# B&R Automation Studio project RobotLineDemo (part 2)

### BRRole.brrole - 5APC4100_TGL4_000/AccessAndSecurity/UserRoleSystem/BRRole.brrole
```
Element BR_Anonymous (Type=BRRole)
Element BR_Engineer (Type=BRRole)
Element BR_Observer (Type=BRRole)
Element BR_SafetyAdmin (Type=BRRole)
Element BR_SecurityAdmin (Type=BRRole)
```

- Physical/Config1/5APC4100_TGL4_000/IoMap.iom: same as Physical/Config1/5APC4100_TGL4_000/Cpu.per
- Physical/Config1/5APC4100_TGL4_000/PvMap.vvm: same as Physical/Config1/5APC4100_TGL4_000/Cpu.per
### Config.mappmotioncfg - 5APC4100_TGL4_000/mappMotion/Config.mappmotioncfg
```
Element MappMotionConfiguration (Type=mappmotioncfg)
  Logger:
    SelectiveLogging = Used
      AdministrativeCommands = Suppressed
      InformationalCommands = Suppressed
  Diagnostics:
    Snapshot = NotUsed
```

### ConvAxes.axis - 5APC4100_TGL4_000/mappMotion/Conveyors/ConvAxes.axis
```
Element gAxis_Conveyor_1 (Type=axis)
  BaseType = LinearPeriodic
    PeriodSettings:
      Period = 4000.0
  MovementLimits:
    Acceleration:
      Acceleration = 1000
    Deceleration:
      Deceleration = 1000
Element gAxis_Conveyor_2 (Type=axis)
  BaseType = LinearPeriodic
    PeriodSettings:
      Period = 4000.0
  MovementLimits:
    Acceleration:
      Acceleration = 1000
    Deceleration:
      Deceleration = 1000
```

### TrkPaths.trackingpath - 5APC4100_TGL4_000/mappMotion/Conveyors/TrkPaths.trackingpath
```
Element gTrkPath_Conveyor_1 (Type=trackingpath)
  Type:
    MaxTrackingFrames = 200
    MaxPositionError = 7.0
    MotionSource = Axis
      AxisRef = gAxis_Conveyor_1
    TrackingFrames:
      AutomaticCreation:
        Condition[1]:
          Distance = 150.0
          Activation = ProcessVariable
            ProcessVariableName = ::MovePrg:Cmd.Details.AutoCreationPath1
          Position:
            Translation:
              X = 0
              Y = -150
        Condition[2]:
          Distance = 150.0
          Activation = ProcessVariable
            ProcessVariableName = ::MovePrg:Cmd.Details.AutoCreationPath1
          Position:
            Translation:
              X = 0
              Y = -75
        Condition[3]:
          Distance = 150.0
          Activation = ProcessVariable
            ProcessVariableName = ::MovePrg:Cmd.Details.AutoCreationPath1
          Position:
            Translation:
              X = 0
              Y = 0
      AutomaticDeletion:
        Condition[1]:
          MinPosition = 0
          MaxPosition = 7000
        Condition[2] = AfterDesynchronization
          AxesGroupRef = gAxesGroup_D4r1100R_1
        Condition[3] = AfterDesynchronization
          AxesGroupRef = gAxesGroup_D4r1100R_2
        Condition[4] = AfterDesynchronization
          AxesGroupRef = gAxesGroup_D4r1100R_3
        Condition[5] = AfterDesynchronization
          AxesGroupRef = gAxesGroup_D4r1100R_4
        Condition[6] = AfterDesynchronization
          AxesGroupRef = gAxesGroup_D4r1100R_5
        Condition[7] = AfterDesynchronization
          AxesGroupRef = gAxesGroup_D4r1100R_6
  SceneViewerObject:
    Frame = Invisible
    Content:
      Template[1]:
        Name = Frame
      Template[2]:
        Name = Product
        VisualRepresentation = 3DMesh
          FileName = Product.tnr
          Material = LightGreyMatte
        Filter[1] = AttributeBased
          Type = ForbiddenBits
            Mask = 2#0000_0000_0000_0000_0000_0000_0000_0001
      Template[3]:
        Name = ProductSelected
        VisualRepresentation = 3DMesh
          FileName = Product.tnr
        Filter[1] = AttributeBased
          Type = MandatoryBits
            Mask = 2#0000_0000_0000_0000_0000_0000_0000_0001
Element gTrkPath_Conveyor_2 (Type=trackingpath)
  Type:
    MaxTrackingFrames = 200
    MaxPositionError = 7.0
    MotionSource = Axis
      AxisRef = gAxis_Conveyor_2
    TrackingFrames:
      AutomaticDeletion:
        Condition[1]:
          MinPosition = -200
          MaxPosition = 7800
  SceneViewerObject:
    Frame = Invisible
    Content:
      Template[1]:
        Name = Frame
      Template[2]:
        Name = Tray
        VisualRepresentation = 3DMesh
          FileName = Tray.tnr
          Material = LightGreyMatte
        Filter[1] = AttributeBased
          Type = MandatoryBits
            Mask = 2#0100_0000_0000
      Template[3]:
        Name = Product
        VisualRepresentation = 3DMesh
          FileName = Product.tnr
          Material = LightGreyMatte
        Filter[1] = AttributeBased
          Type = MandatoryBits
            Mask = 2#0000_0000_0000_0000_0000_1000_0000_0000
```

### Config_1.axesgroup - 5APC4100_TGL4_000/mappMotion/Robots/Codian_D4r1100R_1/Config_1.axesgroup
```
Element gAxesGroup_D4r1100R_1 (Type=axesgroup)  // Codian D4-ST41-1100-R30 [RobotID="CodianD4ST41r1100R30" Version="6.4.1"]
  Type = PathGenAxesGroup
    ProcessingTaskClass = 1
    PhysicalAxes:
      JointAxes:
        JointAxis[1]:
          AxisRef = gAxisQ1_D4r1100R_1
        JointAxis[2]:
          AxisRef = gAxisQ2_D4r1100R_1
        JointAxis[3]:
          AxisRef = gAxisQ3_D4r1100R_1
        JointAxis[4]:
          Name = QC
          AxisRef = gAxisQC_D4r1100R_1
    MechanicalSystem:
      MechSysRef = MechSys_D4r1100R_1
    BasicSettings:
      GeometryPlanning:
        Rounding:
          SymmetricRounding = No
          LastSegment = Whole
          AvoidZeroCurvature = Yes
          NonCartesianRounding = Yes
        MaxTangentialTransitionDeviation = 0.05
      TrajectoryPlanning:
        TorqueLimitConsideration = Approximation
      Miscellaneous:
        TimeStretchOverride:
          JerkSuppression = Basic
            AdaptationTime = 0.3
    StopReaction:
      AxisError:
        AxisReaction = DynamicStop
    AxesGroupFeatures:
      FeatureRef[1] = Feature_Programs_D4r1100R_1
      FeatureRef[2] = Feature_Jogging_D4r1100R_1
      FeatureRef[3] = Feature_FeedForward_D4r1100R_1
      FeatureRef[4] = FrameHierarchyRotBaseAngle1
      FeatureRef[5] = ToolSetup
      FeatureRef[6] = Tracking
      FeatureRef[7] = PathDefinitions
      FeatureRef[8] = Feature_TrkFrmSel_R1
```

### Config_2.axis - 5APC4100_TGL4_000/mappMotion/Robots/Codian_D4r1100R_1/Config_2.axis
```
Element gAxisQ1_D4r1100R_1 (Type=axis)  // Codian D4-ST41-1100-R30 [RobotID="CodianD4ST41r1100R30" Version="6.4.1"]
  BaseTypeIsReadOnly = 1
  BaseType = RotaryBounded
    MeasurementUnitIsReadOnly = 1
    MeasurementResolutionIsReadOnly = 1
    MeasurementResolution = 0.001
    CountDirectionIsReadOnly = 1
    CountDirection = Inverse
  MovementLimitsIsReadOnly = 1
  MovementLimits = InternalForPathControlledAxis
    Position:
      LowerLimitMin = -45.0
      UpperLimitMax = 103.0
      LowerLimit = -45.0
      UpperLimit = 103.0
    VelocityIsReadOnly = 1
    Velocity:
      VelocityMax = 410.0
      Velocity = 410.0
    AccelerationIsReadOnly = 1
    Acceleration:
      AccelerationMax = 25000.0
      Acceleration = 25000.0
    DecelerationIsReadOnly = 1
    Deceleration:
      DecelerationMax = 25000.0
      Deceleration = 25000.0
    JerkIsReadOnly = 1
    Jerk = Advanced
      JerkAccelerationPositiveMin = 0.0
      JerkAccelerationPositiveMax = 5000000.0
      JerkAccelerationPositive = 5000000.0
      JerkAccelerationNegativeMin = 0.0
      JerkAccelerationNegativeMax = 5000000.0
      JerkAccelerationNegative = 5000000.0
      JerkDecelerationPositiveMin = 0.0
      JerkDecelerationPositiveMax = 5000000.0
      JerkDecelerationPositive = 5000000.0
      JerkDecelerationNegativeMin = 0.0
      JerkDecelerationNegativeMax = 5000000.0
      JerkDecelerationNegative = 5000000.0
    TorqueIsReadOnly = 1
    Torque = Basic
      TorqueMax = 15.0
      Torque = 15.0
Element gAxisQ2_D4r1100R_1 (Type=axis)  // Codian D4-ST41-1100-R30 [RobotID="CodianD4ST41r1100R30" Version="6.4.1"]
  BaseTypeIsReadOnly = 1
  BaseType = RotaryBounded
    MeasurementUnitIsReadOnly = 1
    MeasurementResolutionIsReadOnly = 1
    MeasurementResolution = 0.001
    CountDirectionIsReadOnly = 1
    CountDirection = Inverse
  MovementLimitsIsReadOnly = 1
  MovementLimits = InternalForPathControlledAxis
    Position:
      LowerLimitMin = -45.0
      UpperLimitMax = 103.0
      LowerLimit = -45.0
      UpperLimit = 103.0
    VelocityIsReadOnly = 1
    Velocity:
      VelocityMax = 410.0
      Velocity = 410.0
    AccelerationIsReadOnly = 1
    Acceleration:
      AccelerationMax = 25000.0
      Acceleration = 25000.0
    DecelerationIsReadOnly = 1
    Deceleration:
      DecelerationMax = 25000.0
      Deceleration = 25000.0
    JerkIsReadOnly = 1
    Jerk = Advanced
      JerkAccelerationPositiveMin = 0.0
      JerkAccelerationPositiveMax = 5000000.0
      JerkAccelerationPositive = 5000000.0
      JerkAccelerationNegativeMin = 0.0
      JerkAccelerationNegativeMax = 5000000.0
      JerkAccelerationNegative = 5000000.0
      JerkDecelerationPositiveMin = 0.0
      JerkDecelerationPositiveMax = 5000000.0
      JerkDecelerationPositive = 5000000.0
      JerkDecelerationNegativeMin = 0.0
      JerkDecelerationNegativeMax = 5000000.0
      JerkDecelerationNegative = 5000000.0
    TorqueIsReadOnly = 1
    Torque = Basic
      TorqueMax = 15.0
      Torque = 15.0
Element gAxisQ3_D4r1100R_1 (Type=axis)  // Codian D4-ST41-1100-R30 [RobotID="CodianD4ST41r1100R30" Version="6.4.1"]
  BaseTypeIsReadOnly = 1
  BaseType = RotaryBounded
    MeasurementUnitIsReadOnly = 1
    MeasurementResolutionIsReadOnly = 1
    MeasurementResolution = 0.001
    CountDirectionIsReadOnly = 1
    CountDirection = Inverse
  MovementLimitsIsReadOnly = 1
  MovementLimits = InternalForPathControlledAxis
    Position:
      LowerLimitMin = -45.0
      UpperLimitMax = 103.0
      LowerLimit = -45.0
      UpperLimit = 103.0
    VelocityIsReadOnly = 1
    Velocity:
      VelocityMax = 410.0
      Velocity = 410.0
    AccelerationIsReadOnly = 1
    Acceleration:
      AccelerationMax = 25000.0
      Acceleration = 25000.0
    DecelerationIsReadOnly = 1
    Deceleration:
      DecelerationMax = 25000.0
      Deceleration = 25000.0
    JerkIsReadOnly = 1
    Jerk = Advanced
      JerkAccelerationPositiveMin = 0.0
      JerkAccelerationPositiveMax = 5000000.0
      JerkAccelerationPositive = 5000000.0
      JerkAccelerationNegativeMin = 0.0
      JerkAccelerationNegativeMax = 5000000.0
      JerkAccelerationNegative = 5000000.0
      JerkDecelerationPositiveMin = 0.0
      JerkDecelerationPositiveMax = 5000000.0
      JerkDecelerationPositive = 5000000.0
      JerkDecelerationNegativeMin = 0.0
      JerkDecelerationNegativeMax = 5000000.0
      JerkDecelerationNegative = 5000000.0
    TorqueIsReadOnly = 1
    Torque = Basic
      TorqueMax = 15.0
      Torque = 15.0
Element gAxisQC_D4r1100R_1 (Type=axis)  // Codian D4-ST41-1100-R30 [RobotID="CodianD4ST41r1100R30" Version="6.4.1"]
  BaseTypeIsReadOnly = 1
  BaseType = Rotary
    MeasurementUnitIsReadOnly = 1
    MeasurementResolutionIsReadOnly = 1
    MeasurementResolution = 0.001
    CountDirectionIsReadOnly = 1
  MovementLimitsIsReadOnly = 1
  MovementLimits = InternalForPathControlledAxis
    VelocityIsReadOnly = 1
    Velocity:
      VelocityMax = 1150.0
      Velocity = 1150.0
    AccelerationIsReadOnly = 1
    Acceleration:
      AccelerationMax = 28000.0
      Acceleration = 28000.0
    DecelerationIsReadOnly = 1
    Deceleration:
      DecelerationMax = 28000.0
      Deceleration = 28000.0
    JerkIsReadOnly = 1
    Jerk = Advanced
      JerkAccelerationPositiveMin = 0.0
      JerkAccelerationPositiveMax = 4000000.0
      JerkAccelerationPositive = 4000000.0
      JerkAccelerationNegativeMin = 0.0
      JerkAccelerationNegativeMax = 4000000.0
      JerkAccelerationNegative = 4000000.0
      JerkDecelerationPositiveMin = 0.0
      JerkDecelerationPositiveMax = 4000000.0
      JerkDecelerationPositive = 4000000.0
      JerkDecelerationNegativeMin = 0.0
      JerkDecelerationNegativeMax = 4000000.0
      JerkDecelerationNegative = 4000000.0
    TorqueIsReadOnly = 1
    Torque = Basic
      TorqueMax = 9.0
      Torque = 9.0
```

### Config_3.mechanicalsystem - 5APC4100_TGL4_000/mappMotion/Robots/Codian_D4r1100R_1/Config_3.mechanicalsystem
```
Element MechSys_D4r1100R_1 (Type=mechanicalsystem)  // Codian D4-ST41-1100-R30 [RobotID="CodianD4ST41r1100R30" Version="6.4.1"]
  TypeIsReadOnly = 1
  Type = Delta
    SubtypeIsReadOnly = 1
    Subtype = 4AxesDeltaA
      SceneViewerObject = ObjectID
        ID = 2540
      DescriptionIsReadOnly = 1
      Description:
        Dimensions:
          BasePlatform:
            ArmLinkPointIsReadOnly = 1
            Arm1LinkPoint:
              Radius = 207.5
              Z = -110.0
            Arm2LinkPoint:
              Angle = -120.0
              Radius = 207.5
              Z = -110.0
            Arm3LinkPoint:
              Angle = -240.0
              Radius = 207.5
              Z = -110.0
          Arms:
            ArmIsReadOnly = 1
            Arm1:
              UpperArmLength = 320.0
              LowerArmLength = 850.0
            Arm2:
              UpperArmLength = 320.0
              LowerArmLength = 850.0
            Arm3:
              UpperArmLength = 320.0
              LowerArmLength = 850.0
            LowerArmPairDistance = 154.0
          EndEffectorPlatform:
            ArmLinkPointIsReadOnly = 1
            Arm1LinkPoint:
              Radius = 70.0
            Arm2LinkPoint:
              Radius = 70.0
            Arm3LinkPoint:
              Radius = 70.0
            TranslationToFlange:
              Z = -59.0
        Offsets:
          JointAxisIsReadOnly = 1
          JointAxis[1]
          JointAxis[2]
          JointAxis[3]
          JointAxis[4]
        CountDirections:
          JointAxisIsReadOnly = 1
          JointAxis[1]
          JointAxis[2]
          JointAxis[3]
          JointAxis[4]
      TcpOrientation:
        Frames = Used
      WireFrameModel:
        UpperArm1:
          Distance = 5
        LowerArm1:
          Distance = 5
        UpperArm2:
          Distance = 5
        LowerArm2:
          Distance = 5
        UpperArm3:
          Distance = 5
        LowerArm3:
          Distance = 5
        EndEffectorPlatformToFlange:
          Distance = 5
        FlangeToTcp = NotUsed
      DynamicModelIsReadOnly = 1
      InternalDynamicModelIsReadOnly = 1
      InternalDynamicModel = Used
        TypeIsReadOnly = 1
        Type = Codian D4-ST41-1100-R30
        Row[1]:
          Value = 4
          Unit = Variant
          Description = Type of dynamic model
        Row[2]:
          Index = 1
          Value = 2.739
          Unit = 
          Description = m1
        Row[3]:
          Index = 2
          Value = 0.2990988
          Unit = 
          Description = m1*rc1x
        Row[4]:
          Index = 3
          Unit = 
          Description = m1*rc1y
        Row[5]:
          Index = 4
          Value = 0.0257466
          Unit = 
          Description = m1*rc1z
        Row[6]:
          Index = 5
          Unit = 
          Description = m1*rc1x*rc1y
        Row[7]:
          Index = 6
          Unit = 
          Description = m1*rc1y*rc1z
        Row[8]:
          Index = 7
          Value = 0.00281152872
          Unit = 
          Description = m1*rc1x*rc1z
        Row[9]:
          Index = 8
          Value = 0.03266158896
          Unit = 
          Description = m1*rc1x^2
        Row[10]:
          Index = 9
          Unit = 
          Description = m1*rc1y^2
        Row[11]:
          Index = 10
          Value = 0.00024201804
          Unit = 
          Description = m1*rc1z^2
        Row[12]:
          Index = 11
          Unit = 
          Description = Jxx1
        Row[13]:
          Index = 12
          Value = 0.0423
          Unit = 
          Description = Jyy1
        Row[14]:
          Index = 13
          Unit = 
          Description = Jzz1
        Row[15]:
          Index = 14
          Value = 2.739
          Unit = 
          Description = m2
        Row[16]:
          Index = 15
          Value = 0.2990988
          Unit = 
          Description = m2*rc2x
        Row[17]:
          Index = 16
          Unit = 
          Description = m2*rc2y
        Row[18]:
          Index = 17
          Value = 0.0257466
          Unit = 
          Description = m2*rc2z
        Row[19]:
          Index = 18
          Unit = 
          Description = m2*rc2x*rc2y
        Row[20]:
          Index = 19
          Unit = 
          Description = m2*rc2y*rc2z
        Row[21]:
          Index = 20
          Value = 0.00281152872
          Unit = 
          Description = m2*rc2x*rc2z
        Row[22]:
          Index = 21
          Value = 0.03266158896
          Unit = 
          Description = m2*rc2x^2
        Row[23]:
          Index = 22
          Unit = 
          Description = m2*rc2y^2
        Row[24]:
          Index = 23
          Value = 0.00024201804
          Unit = 
          Description = m2*rc2z^2
        Row[25]:
          Index = 24
          Unit = 
          Description = Jxx2
        Row[26]:
          Index = 25
          Value = 0.0423
          Unit = 
          Description = Jyy2
        Row[27]:
          Index = 26
          Unit = 
          Description = Jzz2
        Row[28]:
          Index = 27
          Value = 2.739
          Unit = 
          Description = m3
        Row[29]:
          Index = 28
          Value = 0.2990988
          Unit = 
          Description = m3*rc3x
        Row[30]:
          Index = 29
          Unit = 
          Description = m3*rc3y
        Row[31]:
          Index = 30
          Value = 0.0257466
          Unit = 
          Description = m3*rc3z
        Row[32]:
          Index = 31
          Unit = 
          Description = m3*rc3x*rc3y
        Row[33]:
          Index = 32
          Unit = 
          Description = m3*rc3y*rc3z
        Row[34]:
          Index = 33
          Value = 0.00281152872
          Unit = 
          Description = m3*rc3x*rc3z
        Row[35]:
          Index = 34
          Value = 0.03266158896
          Unit = 
          Description = m3*rc3x^2
        Row[36]:
          Index = 35
          Unit = 
          Description = m3*rc3y^2
        Row[37]:
          Index = 36
          Value = 0.00024201804
          Unit = 
          Description = m3*rc3z^2
        Row[38]:
          Index = 37
          Unit = 
          Description = Jxx3
        Row[39]:
          Index = 38
          Value = 0.0423
          Unit = 
          Description = Jyy3
        Row[40]:
          Index = 39
          Unit = 
          Description = Jzz3
        Row[41]:
          Index = 40
          Value = 0.808
          Unit = 
          Description = m4
        Row[42]:
          Index = 41
          Unit = 
          Description = m4*rc4x
        Row[43]:
          Index = 42
          Unit = 
          Description = m4*rc4y
        Row[44]:
          Index = 43
          Unit = 
          Description = m4*rc4z
        Row[45]:
          Index = 44
          Unit = 
          Description = m4*rc4x*rc4y
        Row[46]:
          Index = 45
          Unit = 
          Description = m4*rc4y*rc4z
        Row[47]:
          Index = 46
          Unit = 
          Description = m4*rc4x*rc4z
        Row[48]:
          Index = 47
          Unit = 
          Description = m4*rc4x^2
        Row[49]:
          Index = 48
          Unit = 
          Description = m4*rc4y^2
        Row[50]:
          Index = 49
          Unit = 
          Description = m4*rc4z^2
        Row[51]:
          Index = 50
          Value = 0.0901
          Unit = 
          Description = Jxx4
        Row[52]:
          Index = 51
          Value = 0.0901
          Unit = 
          Description = Jyy4
        Row[53]:
          Index = 52
          Unit = 
          Description = Jzz4
        Row[54]:
          Index = 53
          Value = 0.808
          Unit = 
          Description = m5
        Row[55]:
          Index = 54
          Unit = 
          Description = m5*rc5x
        Row[56]:
          Index = 55
          Unit = 
          Description = m5*rc5y
        Row[57]:
          Index = 56
          Unit = 
          Description = m5*rc5z
        Row[58]:
          Index = 57
          Unit = 
          Description = m5*rc5x*rc5y
        Row[59]:
          Index = 58
          Unit = 
          Description = m5*rc5y*rc5z
        Row[60]:
          Index = 59
          Unit = 
          Description = m5*rc5x*rc5z
        Row[61]:
          Index = 60
          Unit = 
          Description = m5*rc5x^2
        Row[62]:
          Index = 61
          Unit = 
          Description = m5*rc5y^2
        Row[63]:
          Index = 62
          Unit = 
          Description = m5*rc5z^2
        Row[64]:
          Index = 63
          Value = 0.0901
          Unit = 
          Description = Jxx5
        Row[65]:
          Index = 64
          Value = 0.0901
          Unit = 
          Description = Jyy5
        Row[66]:
          Index = 65
          Unit = 
          Description = Jzz5
        Row[67]:
          Index = 66
          Value = 0.808
          Unit = 
          Description = m6
        Row[68]:
          Index = 67
          Unit = 
          Description = m6*rc6x
        Row[69]:
          Index = 68
          Unit = 
          Description = m6*rc6y
        Row[70]:
          Index = 69
          Unit = 
          Description = m6*rc6z
        Row[71]:
          Index = 70
          Unit = 
          Description = m6*rc6x*rc6y
        Row[72]:
          Index = 71
          Unit = 
          Description = m6*rc6y*rc6z
        Row[73]:
          Index = 72
          Unit = 
          Description = m6*rc6x*rc6z
        Row[74]:
          Index = 73
          Unit = 
          Description = m6*rc6x^2
        Row[75]:
          Index = 74
          Unit = 
          Description = m6*rc6y^2
        Row[76]:
          Index = 75
          Unit = 
          Description = m6*rc6z^2
        Row[77]:
          Index = 76
          Value = 0.0901
          Unit = 
          Description = Jxx6
        Row[78]:
          Index = 77
          Value = 0.0901
          Unit = 
          Description = Jyy6
        Row[79]:
          Index = 78
          Unit = 
          Description = Jzz6
        Row[80]:
          Index = 79
          Value = 2.005
          Unit = 
          Description = m7
        Row[81]:
          Index = 80
          Unit = 
          Description = m7*rc7x
        Row[82]:
          Index = 81
          Unit = 
          Description = m7*rc7y
        Row[83]:
          Index = 82
          Value = 0.47159605
          Unit = 
          Description = m7*rc7z
        Row[84]:
          Index = 83
          Unit = 
          Description = m7*rc7x*rc7y
        Row[85]:
          Index = 84
          Unit = 
          Description = m7*rc7y*rc7z
        Row[86]:
          Index = 85
          Unit = 
          Description = m7*rc7x*rc7z
        Row[87]:
          Index = 86
          Unit = 
          Description = m7*rc7x^2
        Row[88]:
          Index = 87
          Unit = 
          Description = m7*rc7y^2
        Row[89]:
          Index = 88
          Value = 0.110924106921
          Unit = 
          Description = m7*rc7z^2
        Row[90]:
          Index = 89
          Value = 0.071421443
          Unit = 
          Description = Jxx7
        Row[91]:
          Index = 90
          Value = 0.071421443
          Unit = 
          Description = Jyy7
        Row[92]:
          Index = 91
          Value = 0.0003844
          Unit = 
          Description = Jzz7
        Row[93]:
          Index = 92
          Value = 1.8
          Unit = 
          Description = m8
        Row[94]:
          Index = 93
          Unit = 
          Description = m8*rc8x
        Row[95]:
          Index = 94
          Unit = 
          Description = m8*rc8y
        Row[96]:
          Index = 95
          Value = 0.520488
          Unit = 
          Description = m8*rc8z
        Row[97]:
          Index = 96
          Unit = 
          Description = m8*rc8x*rc8y
        Row[98]:
          Index = 97
          Unit = 
          Description = m8*rc8y*rc8z
        Row[99]:
          Index = 98
          Unit = 
          Description = m8*rc8x*rc8z
        Row[100]:
          Index = 99
          Unit = 
          Description = m8*rc8x^2
        Row[101]:
          Index = 100
          Unit = 
          Description = m8*rc8y^2
        Row[102]:
          Index = 101
          Value = 0.15050431008
          Unit = 
          Description = m8*rc8z^2
        Row[103]:
          Index = 102
          Value = 0.093006951
          Unit = 
          Description = Jxx8
        Row[104]:
          Index = 103
          Value = 0.093006951
          Unit = 
          Description = Jyy8
        Row[105]:
          Index = 104
          Value = 0.00097
          Unit = 
          Description = Jzz8
        Row[106]:
          Index = 105
          Value = 2.094
          Unit = 
          Description = m9
        Row[107]:
          Index = 106
          Unit = 
          Description = m9*rc9x
        Row[108]:
          Index = 107
          Unit = 
          Description = m9*rc9y
        Row[109]:
          Index = 108
          Unit = 
          Description = m9*rc9z
        Row[110]:
          Index = 109
          Unit = 
          Description = m9*rc9x*rc9y
        Row[111]:
          Index = 110
          Unit = 
          Description = m9*rc9y*rc9z
        Row[112]:
          Index = 111
          Unit = 
          Description = m9*rc9x*rc9z
        Row[113]:
          Index = 112
          Unit = 
          Description = m9*rc9x^2
        Row[114]:
          Index = 113
          Unit = 
          Description = m9*rc9y^2
        Row[115]:
          Index = 114
          Unit = 
          Description = m9*rc9z^2
        Row[116]:
          Index = 115
          Unit = 
          Description = Jxx9
        Row[117]:
          Index = 116
          Unit = 
          Description = Jyy9
        Row[118]:
          Index = 117
          Unit = 
          Description = Jzz9
        Row[119]:
          Index = 118
          Unit = 
          Description = m10
        Row[120]:
          Index = 119
          Unit = 
          Description = m10*rc10x
        Row[121]:
          Index = 120
          Unit = 
          Description = m10*rc10y
        Row[122]:
          Index = 121
          Unit = 
          Description = m10*rc10z
        Row[123]:
          Index = 122
          Unit = 
          Description = m10*rc10x*rc10y
        Row[124]:
          Index = 123
          Unit = 
          Description = m10*rc10y*rc10z
        Row[125]:
          Index = 124
          Unit = 
          Description = m10*rc10x*rc10z
        Row[126]:
          Index = 125
          Unit = 
          Description = m10*rc10x^2
        Row[127]:
          Index = 126
          Unit = 
          Description = m10*rc10y^2
        Row[128]:
          Index = 127
          Unit = 
          Description = m10*rc10z^2
        Row[129]:
          Index = 128
          Unit = 
          Description = Jxx10
        Row[130]:
          Index = 129
          Unit = 
          Description = Jyy10
        Row[131]:
          Index = 130
          Value = 0.0001507
          Unit = 
          Description = Jzz10
        Row[132]:
          Index = 144
          Value = 0.0005703
          Unit = 
          Description = JDrive1
        Row[133]:
          Index = 145
          Value = 0.0005703
          Unit = 
          Description = JDrive2
        Row[134]:
          Index = 146
          Value = 0.0005703
          Unit = 
          Description = JDrive3
        Row[135]:
          Index = 147
          Value = 0.0001462
          Unit = 
          Description = JDrive4
        Row[136]:
          Index = 148
          Value = 2.35907414398
          Unit = 
          Description = dV1
        Row[137]:
          Index = 149
          Value = 2.35907414398
          Unit = 
          Description = dV2
        Row[138]:
          Index = 150
          Value = 2.35907414398
          Unit = 
          Description = dV3
        Row[139]:
          Index = 151
          Value = 0.0159154943092
          Unit = 
          Description = dV4
        Row[140]:
          Index = 152
          Value = 4.235
          Unit = 
          Description = dC1
        Row[141]:
          Index = 153
          Value = 4.235
          Unit = 
          Description = dC2
        Row[142]:
          Index = 154
          Value = 4.235
          Unit = 
          Description = dC3
        Row[143]:
          Index = 155
          Value = 1.0
          Unit = 
          Description = dC4
      InternalDynamicLimits = Used
        TypeIsReadOnly = 1
        Type = Codian D4-ST41-1100-R30
        GearboxLimits:
          Row[1]:
            Value = 4
            Unit = Variant
            Description = Type of dynamic model
          Row[2]:
            Index = 1
            Value = 370.0
            Unit = Nm
            Description = Gearbox Drive 1 Output Torque Limit
          Row[3]:
            Index = 2
            Value = 370.0
            Unit = Nm
            Description = Gearbox Drive 2 Output Torque Limit
          Row[4]:
            Index = 3
            Value = 370.0
            Unit = Nm
            Description = Gearbox Drive 3 Output Torque Limit
          Row[5]:
            Index = 4
            Value = 17.0
            Unit = Nm
            Description = Gearbox Drive 4 Output Torque Limit
        CrossSectionLimits:
          Row[1]:
            Value = 4
            Unit = Variant
            Description = Type of dynamic model
          Row[2]:
            Index = 1
            Value = 10000.0
            Unit = N
            Description = 
          Row[3]:
            Index = 2
            Value = 10000.0
            Unit = N
            Description = 
          Row[4]:
            Index = 3
            Value = 10000.0
            Unit = N
            Description = 
          Row[5]:
            Index = 4
            Value = 141.0
            Unit = Nm
            Description = 
          Row[6]:
            Index = 5
            Value = 141.0
            Unit = Nm
            Description = 
          Row[7]:
            Index = 6
            Value = 10000.0
            Unit = Nm
            Description = 
          Row[8]:
            Index = 7
            Value = 750.0
            Unit = N
            Description = 
          Row[9]:
            Index = 8
            Value = 750.0
            Unit = N
            Description = 
          Row[10]:
            Index = 9
            Value = 750.0
            Unit = N
            Description = 
          Row[11]:
            Index = 10
            Value = 750.0
            Unit = N
            Description = 
          Row[12]:
            Index = 11
            Value = 750.0
            Unit = N
            Description = 
          Row[13]:
            Index = 12
            Value = 750.0
            Unit = N
            Description = 
      LoadDependentJerkLimitsIsReadOnly = 1
      LoadDependentJerkLimits = PayloadDependentJerkReduction
        JerkReduction[1]:
          PayloadInKgIsReadOnly = 1
          PayloadInKg = 0.0
          JerkReductionInPercentIsReadOnly = 1
          JerkReductionInPercent = 0.0
        JerkReduction[2]:
          PayloadInKgIsReadOnly = 1
          PayloadInKg = 7.0
          JerkReductionInPercentIsReadOnly = 1
          JerkReductionInPercent = 20.0
        JerkReduction[3]:
          PayloadInKgIsReadOnly = 1
          PayloadInKg = 13.0
          JerkReductionInPercentIsReadOnly = 1
          JerkReductionInPercent = 60.0
        JerkReduction[4]:
          PayloadInKgIsReadOnly = 1
          PayloadInKg = 19.0
          JerkReductionInPercentIsReadOnly = 1
          JerkReductionInPercent = 60.0
        JerkReduction[5]:
          PayloadInKgIsReadOnly = 1
          PayloadInKg = 23.0
          JerkReductionInPercentIsReadOnly = 1
          JerkReductionInPercent = 80.0
      JointAxesPositionLimits:
        JointAxisIsReadOnly = 1
        JointAxis[1]
        JointAxis[2]
        JointAxis[3]
        JointAxis[4]
      WorkingRangeIsReadOnly = 1
      WorkingRange = Extended
        MainCylinderDiameterIsReadOnly = 1
        MainCylinderDiameter = 1100.0
        BaseToTopConeIsReadOnly = 1
        BaseToTopCone = 735.0
        MainCylinderOffsetIsReadOnly = 1
        MainCylinderOffset = 270.0
        MainConeOffsetIsReadOnly = 1
        MainConeOffset = 350.0
        BottomConeOffsetIsReadOnly = 1
        BottomConeOffset = 420.0
        MainConeDiameterIsReadOnly = 1
        MainConeDiameter = 820.0
        BottomConeDiameterIsReadOnly = 1
        BottomConeDiameter = 340.0
        TopConeOffsetIsReadOnly = 1
        TopConeDiameterIsReadOnly = 1
        TopConeDiameter = 1100.0
```

### Config_4.axesgroupfeature - 5APC4100_TGL4_000/mappMotion/Robots/Codian_D4r1100R_1/Config_4.axesgroupfeature
```
Element Feature_TrkFrmSel_R1 (Type=axesgroupfeature)
  Type = TrackingFrameSelection
    Selectors:
      Selector[1]:
        Name = ProductSelector
        Strategy = MinimumDistanceToPoint
          Origin = MCS
            Translation:
              X = -350
              Y = 300
        Filters:
          Filter[1]:
            TrackingPathRef[1] = gTrkPath_Conveyor_1
          Filter[2] = SelectionArea
            Area[1] = Cylinder
              Origin = MCS
              Translation:
                X = -470
                Z = -100
              Dimensions:
                Radius = 475
                Height = 250
        LockingAfterSelection = AllSelectors
      Selector[2]:
        Name = PlacePositionSelector
        Strategy = MaximumXValueOnTrackingPath
        Filters:
          Filter[1]:
            TrackingPathRef[1] = gTrkPath_Conveyor_2
          Filter[2] = SelectionArea
            Area[1] = Cylinder
              Origin = MCS
              Translation:
                X = 250
                Z = -100
              Dimensions:
                Radius = 500
                Height = 250
        LockingAfterSelection = AllSelectors
      Selector[3]:
        Name = PlacePositionSelectorPrior
        Strategy = MaximumXValueOnTrackingPath
        Filters:
          Filter[1]:
            TrackingPathRef[1] = gTrkPath_Conveyor_2
          Filter[2] = SelectionArea
            Area[1]:
              Origin = MCS
              Translation:
                X = -300
                Y = 200
                Z = -100
              Dimensions:
                Length = 700
                Width = 200
                Height = 250
        LockingAfterSelection = AllSelectors
Element Feature_Programs_D4r1100R_1 (Type=axesgroupfeature)  // Codian D4-ST41-1100-R30 [RobotID="CodianD4ST41r1100R30" Version="6.4.1"]
  Type:
    InitialSettings:
      AccuracyHoldDelays = User defined
        UserAxesDelay = 0.06
    ProgramElements:
      PVs:
        PV[1]:
          PvName = ::MovePrg:GripperRobot1OpenClose
          Advanced:
            Alias = CloseGripper
            Synchronization = Path
Element Feature_Jogging_D4r1100R_1 (Type=axesgroupfeature)  // Codian D4-ST41-1100-R30 [RobotID="CodianD4ST41r1100R30" Version="6.4.1"]
  Type = Jogging
Element Feature_FeedForward_D4r1100R_1 (Type=axesgroupfeature)  // Codian D4-ST41-1100-R30 [RobotID="CodianD4ST41r1100R30" Version="6.4.1"]
  Type = FeedForward
    RiseTime = 0.25
    Filter = AxisJerkTime
```

### Config_5.axesgroup - 5APC4100_TGL4_000/mappMotion/Robots/Codian_D4r1100R_2/Config_5.axesgroup
```
Element gAxesGroup_D4r1100R_2 (Type=axesgroup)  // Codian D4-ST41-1100-R30 [RobotID="CodianD4ST41r1100R30" Version="6.4.1"]
  Type = PathGenAxesGroup
    ProcessingTaskClass = 1
    PhysicalAxes:
      JointAxes:
        JointAxis[1]:
          AxisRef = gAxisQ1_D4r1100R_2
        JointAxis[2]:
          AxisRef = gAxisQ2_D4r1100R_2
        JointAxis[3]:
          AxisRef = gAxisQ3_D4r1100R_2
        JointAxis[4]:
          Name = QC
          AxisRef = gAxisQC_D4r1100R_2
    MechanicalSystem:
      MechSysRef = MechSys_D4r1100R_2
    BasicSettings:
      GeometryPlanning:
        Rounding:
          SymmetricRounding = No
          LastSegment = Whole
          AvoidZeroCurvature = Yes
          NonCartesianRounding = Yes
        MaxTangentialTransitionDeviation = 0.05
      TrajectoryPlanning:
        TorqueLimitConsideration = Approximation
      Miscellaneous:
        TimeStretchOverride:
          JerkSuppression = Basic
            AdaptationTime = 0.3
    StopReaction:
      AxisError:
        AxisReaction = DynamicStop
    AxesGroupFeatures:
      FeatureRef[1] = Feature_Programs_D4r1100R_2
      FeatureRef[2] = Feature_Jogging_D4r1100R_2
      FeatureRef[3] = Feature_FeedForward_D4r1100R_2
      FeatureRef[4] = FrameHierarchyRotBaseAngle2
      FeatureRef[5] = ToolSetup
      FeatureRef[6] = Tracking
      FeatureRef[7] = PathDefinitions
      FeatureRef[8] = Feature_TrkFrmSel_R2
```

### Config_6.axis - 5APC4100_TGL4_000/mappMotion/Robots/Codian_D4r1100R_2/Config_6.axis
```
Element gAxisQ1_D4r1100R_2 (Type=axis)  // Codian D4-ST41-1100-R30 [RobotID="CodianD4ST41r1100R30" Version="6.4.1"]
  BaseTypeIsReadOnly = 1
  BaseType = RotaryBounded
    MeasurementUnitIsReadOnly = 1
    MeasurementResolutionIsReadOnly = 1
    MeasurementResolution = 0.001
    CountDirectionIsReadOnly = 1
    CountDirection = Inverse
  MovementLimitsIsReadOnly = 1
  MovementLimits = InternalForPathControlledAxis
    Position:
      LowerLimitMin = -45.0
      UpperLimitMax = 103.0
      LowerLimit = -45.0
      UpperLimit = 103.0
    VelocityIsReadOnly = 1
    Velocity:
      VelocityMax = 410.0
      Velocity = 410.0
    AccelerationIsReadOnly = 1
    Acceleration:
      AccelerationMax = 25000.0
      Acceleration = 25000.0
    DecelerationIsReadOnly = 1
    Deceleration:
      DecelerationMax = 25000.0
      Deceleration = 25000.0
    JerkIsReadOnly = 1
    Jerk = Advanced
      JerkAccelerationPositiveMin = 0.0
      JerkAccelerationPositiveMax = 5000000.0
      JerkAccelerationPositive = 5000000.0
      JerkAccelerationNegativeMin = 0.0
      JerkAccelerationNegativeMax = 5000000.0
      JerkAccelerationNegative = 5000000.0
      JerkDecelerationPositiveMin = 0.0
      JerkDecelerationPositiveMax = 5000000.0
      JerkDecelerationPositive = 5000000.0
      JerkDecelerationNegativeMin = 0.0
      JerkDecelerationNegativeMax = 5000000.0
      JerkDecelerationNegative = 5000000.0
    TorqueIsReadOnly = 1
    Torque = Basic
      TorqueMax = 15.0
      Torque = 15.0
Element gAxisQ2_D4r1100R_2 (Type=axis)  // Codian D4-ST41-1100-R30 [RobotID="CodianD4ST41r1100R30" Version="6.4.1"]
  BaseTypeIsReadOnly = 1
  BaseType = RotaryBounded
    MeasurementUnitIsReadOnly = 1
    MeasurementResolutionIsReadOnly = 1
    MeasurementResolution = 0.001
    CountDirectionIsReadOnly = 1
    CountDirection = Inverse
  MovementLimitsIsReadOnly = 1
  MovementLimits = InternalForPathControlledAxis
    Position:
      LowerLimitMin = -45.0
      UpperLimitMax = 103.0
      LowerLimit = -45.0
      UpperLimit = 103.0
    VelocityIsReadOnly = 1
    Velocity:
      VelocityMax = 410.0
      Velocity = 410.0
    AccelerationIsReadOnly = 1
    Acceleration:
      AccelerationMax = 25000.0
      Acceleration = 25000.0
    DecelerationIsReadOnly = 1
    Deceleration:
      DecelerationMax = 25000.0
      Deceleration = 25000.0
    JerkIsReadOnly = 1
    Jerk = Advanced
      JerkAccelerationPositiveMin = 0.0
      JerkAccelerationPositiveMax = 5000000.0
      JerkAccelerationPositive = 5000000.0
      JerkAccelerationNegativeMin = 0.0
      JerkAccelerationNegativeMax = 5000000.0
      JerkAccelerationNegative = 5000000.0
      JerkDecelerationPositiveMin = 0.0
      JerkDecelerationPositiveMax = 5000000.0
      JerkDecelerationPositive = 5000000.0
      JerkDecelerationNegativeMin = 0.0
      JerkDecelerationNegativeMax = 5000000.0
      JerkDecelerationNegative = 5000000.0
    TorqueIsReadOnly = 1
    Torque = Basic
      TorqueMax = 15.0
      Torque = 15.0
Element gAxisQ3_D4r1100R_2 (Type=axis)  // Codian D4-ST41-1100-R30 [RobotID="CodianD4ST41r1100R30" Version="6.4.1"]
  BaseTypeIsReadOnly = 1
  BaseType = RotaryBounded
    MeasurementUnitIsReadOnly = 1
    MeasurementResolutionIsReadOnly = 1
    MeasurementResolution = 0.001
    CountDirectionIsReadOnly = 1
    CountDirection = Inverse
  MovementLimitsIsReadOnly = 1
  MovementLimits = InternalForPathControlledAxis
    Position:
      LowerLimitMin = -45.0
      UpperLimitMax = 103.0
      LowerLimit = -45.0
      UpperLimit = 103.0
    VelocityIsReadOnly = 1
    Velocity:
      VelocityMax = 410.0
      Velocity = 410.0
    AccelerationIsReadOnly = 1
    Acceleration:
      AccelerationMax = 25000.0
      Acceleration = 25000.0
    DecelerationIsReadOnly = 1
    Deceleration:
      DecelerationMax = 25000.0
      Deceleration = 25000.0
    JerkIsReadOnly = 1
    Jerk = Advanced
      JerkAccelerationPositiveMin = 0.0
      JerkAccelerationPositiveMax = 5000000.0
      JerkAccelerationPositive = 5000000.0
      JerkAccelerationNegativeMin = 0.0
      JerkAccelerationNegativeMax = 5000000.0
      JerkAccelerationNegative = 5000000.0
      JerkDecelerationPositiveMin = 0.0
      JerkDecelerationPositiveMax = 5000000.0
      JerkDecelerationPositive = 5000000.0
      JerkDecelerationNegativeMin = 0.0
      JerkDecelerationNegativeMax = 5000000.0
      JerkDecelerationNegative = 5000000.0
    TorqueIsReadOnly = 1
    Torque = Basic
      TorqueMax = 15.0
      Torque = 15.0
Element gAxisQC_D4r1100R_2 (Type=axis)  // Codian D4-ST41-1100-R30 [RobotID="CodianD4ST41r1100R30" Version="6.4.1"]
  BaseTypeIsReadOnly = 1
  BaseType = Rotary
    MeasurementUnitIsReadOnly = 1
    MeasurementResolutionIsReadOnly = 1
    MeasurementResolution = 0.001
    CountDirectionIsReadOnly = 1
  MovementLimitsIsReadOnly = 1
  MovementLimits = InternalForPathControlledAxis
    VelocityIsReadOnly = 1
    Velocity:
      VelocityMax = 1150.0
      Velocity = 1150.0
    AccelerationIsReadOnly = 1
    Acceleration:
      AccelerationMax = 28000.0
      Acceleration = 28000.0
    DecelerationIsReadOnly = 1
    Deceleration:
      DecelerationMax = 28000.0
      Deceleration = 28000.0
    JerkIsReadOnly = 1
    Jerk = Advanced
      JerkAccelerationPositiveMin = 0.0
      JerkAccelerationPositiveMax = 4000000.0
      JerkAccelerationPositive = 4000000.0
      JerkAccelerationNegativeMin = 0.0
      JerkAccelerationNegativeMax = 4000000.0
      JerkAccelerationNegative = 4000000.0
      JerkDecelerationPositiveMin = 0.0
      JerkDecelerationPositiveMax = 4000000.0
      JerkDecelerationPositive = 4000000.0
      JerkDecelerationNegativeMin = 0.0
      JerkDecelerationNegativeMax = 4000000.0
      JerkDecelerationNegative = 4000000.0
    TorqueIsReadOnly = 1
    Torque = Basic
      TorqueMax = 9.0
      Torque = 9.0
```

### Config_7.mechanicalsystem - 5APC4100_TGL4_000/mappMotion/Robots/Codian_D4r1100R_2/Config_7.mechanicalsystem
```
Element MechSys_D4r1100R_2 (Type=mechanicalsystem)  // Codian D4-ST41-1100-R30 [RobotID="CodianD4ST41r1100R30" Version="6.4.1"]
  TypeIsReadOnly = 1
  Type = Delta
    SubtypeIsReadOnly = 1
    Subtype = 4AxesDeltaA
      SceneViewerObject = ObjectID
        ID = 2540
      DescriptionIsReadOnly = 1
      Description:
        Dimensions:
          BasePlatform:
            ArmLinkPointIsReadOnly = 1
            Arm1LinkPoint:
              Radius = 207.5
              Z = -110.0
            Arm2LinkPoint:
              Angle = -120.0
              Radius = 207.5
              Z = -110.0
            Arm3LinkPoint:
              Angle = -240.0
              Radius = 207.5
              Z = -110.0
          Arms:
            ArmIsReadOnly = 1
            Arm1:
              UpperArmLength = 320.0
              LowerArmLength = 850.0
            Arm2:
              UpperArmLength = 320.0
              LowerArmLength = 850.0
            Arm3:
              UpperArmLength = 320.0
              LowerArmLength = 850.0
            LowerArmPairDistance = 154.0
          EndEffectorPlatform:
            ArmLinkPointIsReadOnly = 1
            Arm1LinkPoint:
              Radius = 70.0
            Arm2LinkPoint:
              Radius = 70.0
            Arm3LinkPoint:
              Radius = 70.0
            TranslationToFlange:
              Z = -59.0
        Offsets:
          JointAxisIsReadOnly = 1
          JointAxis[1]
          JointAxis[2]
          JointAxis[3]
          JointAxis[4]
        CountDirections:
          JointAxisIsReadOnly = 1
          JointAxis[1]
          JointAxis[2]
          JointAxis[3]
          JointAxis[4]
      TcpOrientation:
        Frames = Used
      WireFrameModel:
        UpperArm1:
          Distance = 5
        LowerArm1:
          Distance = 5
        UpperArm2:
          Distance = 5
        LowerArm2:
          Distance = 5
        UpperArm3:
          Distance = 5
        LowerArm3:
          Distance = 5
        EndEffectorPlatformToFlange:
          Distance = 5
        FlangeToTcp = NotUsed
      DynamicModelIsReadOnly = 1
      InternalDynamicModelIsReadOnly = 1
      InternalDynamicModel = Used
        TypeIsReadOnly = 1
        Type = Codian D4-ST41-1100-R30
        Row[1]:
          Value = 4
          Unit = Variant
          Description = Type of dynamic model
        Row[2]:
          Index = 1
          Value = 2.739
          Unit = 
          Description = m1
        Row[3]:
          Index = 2
          Value = 0.2990988
          Unit = 
          Description = m1*rc1x
        Row[4]:
          Index = 3
          Unit = 
          Description = m1*rc1y
        Row[5]:
          Index = 4
          Value = 0.0257466
          Unit = 
          Description = m1*rc1z
        Row[6]:
          Index = 5
          Unit = 
          Description = m1*rc1x*rc1y
        Row[7]:
          Index = 6
          Unit = 
          Description = m1*rc1y*rc1z
        Row[8]:
          Index = 7
          Value = 0.00281152872
          Unit = 
          Description = m1*rc1x*rc1z
        Row[9]:
          Index = 8
          Value = 0.03266158896
          Unit = 
          Description = m1*rc1x^2
        Row[10]:
          Index = 9
          Unit = 
          Description = m1*rc1y^2
        Row[11]:
          Index = 10
          Value = 0.00024201804
          Unit = 
          Description = m1*rc1z^2
        Row[12]:
          Index = 11
          Unit = 
          Description = Jxx1
        Row[13]:
          Index = 12
          Value = 0.0423
          Unit = 
          Description = Jyy1
        Row[14]:
          Index = 13
          Unit = 
          Description = Jzz1
        Row[15]:
          Index = 14
          Value = 2.739
          Unit = 
          Description = m2
        Row[16]:
          Index = 15
          Value = 0.2990988
          Unit = 
          Description = m2*rc2x
        Row[17]:
          Index = 16
          Unit = 
          Description = m2*rc2y
        Row[18]:
          Index = 17
          Value = 0.0257466
          Unit = 
          Description = m2*rc2z
        Row[19]:
          Index = 18
          Unit = 
          Description = m2*rc2x*rc2y
        Row[20]:
          Index = 19
          Unit = 
          Description = m2*rc2y*rc2z
        Row[21]:
          Index = 20
          Value = 0.00281152872
          Unit = 
          Description = m2*rc2x*rc2z
        Row[22]:
          Index = 21
          Value = 0.03266158896
          Unit = 
          Description = m2*rc2x^2
        Row[23]:
          Index = 22
          Unit = 
          Description = m2*rc2y^2
        Row[24]:
          Index = 23
          Value = 0.00024201804
          Unit = 
          Description = m2*rc2z^2
        Row[25]:
          Index = 24
          Unit = 
          Description = Jxx2
        Row[26]:
          Index = 25
          Value = 0.0423
          Unit = 
          Description = Jyy2
        Row[27]:
          Index = 26
          Unit = 
          Description = Jzz2
        Row[28]:
          Index = 27
          Value = 2.739
          Unit = 
          Description = m3
        Row[29]:
          Index = 28
          Value = 0.2990988
          Unit = 
          Description = m3*rc3x
        Row[30]:
          Index = 29
          Unit = 
          Description = m3*rc3y
        Row[31]:
          Index = 30
          Value = 0.0257466
          Unit = 
          Description = m3*rc3z
        Row[32]:
          Index = 31
          Unit = 
          Description = m3*rc3x*rc3y
        Row[33]:
          Index = 32
          Unit = 
          Description = m3*rc3y*rc3z
        Row[34]:
          Index = 33
          Value = 0.00281152872
          Unit = 
          Description = m3*rc3x*rc3z
        Row[35]:
          Index = 34
          Value = 0.03266158896
          Unit = 
          Description = m3*rc3x^2
        Row[36]:
          Index = 35
          Unit = 
          Description = m3*rc3y^2
        Row[37]:
          Index = 36
          Value = 0.00024201804
          Unit = 
          Description = m3*rc3z^2
        Row[38]:
          Index = 37
          Unit = 
          Description = Jxx3
        Row[39]:
          Index = 38
          Value = 0.0423
          Unit = 
          Description = Jyy3
        Row[40]:
          Index = 39
          Unit = 
          Description = Jzz3
        Row[41]:
          Index = 40
          Value = 0.808
          Unit = 
          Description = m4
        Row[42]:
          Index = 41
          Unit = 
          Description = m4*rc4x
        Row[43]:
          Index = 42
          Unit = 
          Description = m4*rc4y
        Row[44]:
          Index = 43
          Unit = 
          Description = m4*rc4z
        Row[45]:
          Index = 44
          Unit = 
          Description = m4*rc4x*rc4y
        Row[46]:
          Index = 45
          Unit = 
          Description = m4*rc4y*rc4z
        Row[47]:
          Index = 46
          Unit = 
          Description = m4*rc4x*rc4z
        Row[48]:
          Index = 47
          Unit = 
          Description = m4*rc4x^2
        Row[49]:
          Index = 48
          Unit = 
          Description = m4*rc4y^2
        Row[50]:
          Index = 49
          Unit = 
          Description = m4*rc4z^2
        Row[51]:
          Index = 50
          Value = 0.0901
          Unit = 
          Description = Jxx4
        Row[52]:
          Index = 51
          Value = 0.0901
          Unit = 
          Description = Jyy4
        Row[53]:
          Index = 52
          Unit = 
          Description = Jzz4
        Row[54]:
          Index = 53
          Value = 0.808
          Unit = 
          Description = m5
        Row[55]:
          Index = 54
          Unit = 
          Description = m5*rc5x
        Row[56]:
          Index = 55
          Unit = 
          Description = m5*rc5y
        Row[57]:
          Index = 56
          Unit = 
          Description = m5*rc5z
        Row[58]:
          Index = 57
          Unit = 
          Description = m5*rc5x*rc5y
        Row[59]:
          Index = 58
          Unit = 
          Description = m5*rc5y*rc5z
        Row[60]:
          Index = 59
          Unit = 
          Description = m5*rc5x*rc5z
        Row[61]:
          Index = 60
          Unit = 
          Description = m5*rc5x^2
        Row[62]:
          Index = 61
          Unit = 
          Description = m5*rc5y^2
        Row[63]:
          Index = 62
          Unit = 
          Description = m5*rc5z^2
        Row[64]:
          Index = 63
          Value = 0.0901
          Unit = 
          Description = Jxx5
        Row[65]:
          Index = 64
          Value = 0.0901
          Unit = 
          Description = Jyy5
        Row[66]:
          Index = 65
          Unit = 
          Description = Jzz5
        Row[67]:
          Index = 66
          Value = 0.808
          Unit = 
          Description = m6
        Row[68]:
          Index = 67
          Unit = 
          Description = m6*rc6x
        Row[69]:
          Index = 68
          Unit = 
          Description = m6*rc6y
        Row[70]:
          Index = 69
          Unit = 
          Description = m6*rc6z
        Row[71]:
          Index = 70
          Unit = 
          Description = m6*rc6x*rc6y
        Row[72]:
          Index = 71
          Unit = 
          Description = m6*rc6y*rc6z
        Row[73]:
          Index = 72
          Unit = 
          Description = m6*rc6x*rc6z
        Row[74]:
          Index = 73
          Unit = 
          Description = m6*rc6x^2
        Row[75]:
          Index = 74
          Unit = 
          Description = m6*rc6y^2
        Row[76]:
          Index = 75
          Unit = 
          Description = m6*rc6z^2
        Row[77]:
          Index = 76
          Value = 0.0901
          Unit = 
          Description = Jxx6
        Row[78]:
          Index = 77
          Value = 0.0901
          Unit = 
          Description = Jyy6
        Row[79]:
          Index = 78
          Unit = 
          Description = Jzz6
        Row[80]:
          Index = 79
          Value = 2.005
          Unit = 
          Description = m7
        Row[81]:
          Index = 80
          Unit = 
          Description = m7*rc7x
        Row[82]:
          Index = 81
          Unit = 
          Description = m7*rc7y
        Row[83]:
          Index = 82
          Value = 0.47159605
          Unit = 
          Description = m7*rc7z
        Row[84]:
          Index = 83
          Unit = 
          Description = m7*rc7x*rc7y
        Row[85]:
          Index = 84
          Unit = 
          Description = m7*rc7y*rc7z
        Row[86]:
          Index = 85
          Unit = 
          Description = m7*rc7x*rc7z
        Row[87]:
          Index = 86
          Unit = 
          Description = m7*rc7x^2
        Row[88]:
          Index = 87
          Unit = 
          Description = m7*rc7y^2
        Row[89]:
          Index = 88
          Value = 0.110924106921
          Unit = 
          Description = m7*rc7z^2
        Row[90]:
          Index = 89
          Value = 0.071421443
          Unit = 
          Description = Jxx7
        Row[91]:
          Index = 90
          Value = 0.071421443
          Unit = 
          Description = Jyy7
        Row[92]:
          Index = 91
          Value = 0.0003844
          Unit = 
          Description = Jzz7
        Row[93]:
          Index = 92
          Value = 1.8
          Unit = 
          Description = m8
        Row[94]:
          Index = 93
          Unit = 
          Description = m8*rc8x
        Row[95]:
          Index = 94
          Unit = 
          Description = m8*rc8y
        Row[96]:
          Index = 95
          Value = 0.520488
          Unit = 
          Description = m8*rc8z
        Row[97]:
          Index = 96
          Unit = 
          Description = m8*rc8x*rc8y
        Row[98]:
          Index = 97
          Unit = 
          Description = m8*rc8y*rc8z
        Row[99]:
          Index = 98
          Unit = 
          Description = m8*rc8x*rc8z
        Row[100]:
          Index = 99
          Unit = 
          Description = m8*rc8x^2
        Row[101]:
          Index = 100
          Unit = 
          Description = m8*rc8y^2
        Row[102]:
          Index = 101
          Value = 0.15050431008
          Unit = 
          Description = m8*rc8z^2
        Row[103]:
          Index = 102
          Value = 0.093006951
          Unit = 
          Description = Jxx8
        Row[104]:
          Index = 103
          Value = 0.093006951
          Unit = 
          Description = Jyy8
        Row[105]:
          Index = 104
          Value = 0.00097
          Unit = 
          Description = Jzz8
        Row[106]:
          Index = 105
          Value = 2.094
          Unit = 
          Description = m9
        Row[107]:
          Index = 106
          Unit = 
          Description = m9*rc9x
        Row[108]:
          Index = 107
          Unit = 
          Description = m9*rc9y
        Row[109]:
          Index = 108
          Unit = 
          Description = m9*rc9z
        Row[110]:
          Index = 109
          Unit = 
          Description = m9*rc9x*rc9y
        Row[111]:
          Index = 110
          Unit = 
          Description = m9*rc9y*rc9z
        Row[112]:
          Index = 111
          Unit = 
          Description = m9*rc9x*rc9z
        Row[113]:
          Index = 112
          Unit = 
          Description = m9*rc9x^2
        Row[114]:
          Index = 113
          Unit = 
          Description = m9*rc9y^2
        Row[115]:
          Index = 114
          Unit = 
          Description = m9*rc9z^2
        Row[116]:
          Index = 115
          Unit = 
          Description = Jxx9
        Row[117]:
          Index = 116
          Unit = 
          Description = Jyy9
        Row[118]:
          Index = 117
          Unit = 
          Description = Jzz9
        Row[119]:
          Index = 118
          Unit = 
          Description = m10
        Row[120]:
          Index = 119
          Unit = 
          Description = m10*rc10x
        Row[121]:
          Index = 120
          Unit = 
          Description = m10*rc10y
        Row[122]:
          Index = 121
          Unit = 
          Description = m10*rc10z
        Row[123]:
          Index = 122
          Unit = 
          Description = m10*rc10x*rc10y
        Row[124]:
          Index = 123
          Unit = 
          Description = m10*rc10y*rc10z
        Row[125]:
          Index = 124
          Unit = 
          Description = m10*rc10x*rc10z
        Row[126]:
          Index = 125
          Unit = 
          Description = m10*rc10x^2
        Row[127]:
          Index = 126
          Unit = 
          Description = m10*rc10y^2
        Row[128]:
          Index = 127
          Unit = 
          Description = m10*rc10z^2
        Row[129]:
          Index = 128
          Unit = 
          Description = Jxx10
        Row[130]:
          Index = 129
          Unit = 
          Description = Jyy10
        Row[131]:
          Index = 130
          Value = 0.0001507
          Unit = 
          Description = Jzz10
        Row[132]:
          Index = 144
          Value = 0.0005703
          Unit = 
          Description = JDrive1
        Row[133]:
          Index = 145
          Value = 0.0005703
          Unit = 
          Description = JDrive2
        Row[134]:
          Index = 146
          Value = 0.0005703
          Unit = 
          Description = JDrive3
        Row[135]:
          Index = 147
          Value = 0.0001462
          Unit = 
          Description = JDrive4
        Row[136]:
          Index = 148
          Value = 2.35907414398
          Unit = 
          Description = dV1
        Row[137]:
          Index = 149
          Value = 2.35907414398
          Unit = 
          Description = dV2
        Row[138]:
          Index = 150
          Value = 2.35907414398
          Unit = 
          Description = dV3
        Row[139]:
          Index = 151
          Value = 0.0159154943092
          Unit = 
          Description = dV4
        Row[140]:
          Index = 152
          Value = 4.235
          Unit = 
          Description = dC1
        Row[141]:
          Index = 153
          Value = 4.235
          Unit = 
          Description = dC2
        Row[142]:
          Index = 154
          Value = 4.235
          Unit = 
          Description = dC3
        Row[143]:
          Index = 155
          Value = 1.0
          Unit = 
          Description = dC4
      InternalDynamicLimits = Used
        TypeIsReadOnly = 1
        Type = Codian D4-ST41-1100-R30
        GearboxLimits:
          Row[1]:
            Value = 4
            Unit = Variant
            Description = Type of dynamic model
          Row[2]:
            Index = 1
            Value = 370.0
            Unit = Nm
            Description = Gearbox Drive 1 Output Torque Limit
          Row[3]:
            Index = 2
            Value = 370.0
            Unit = Nm
            Description = Gearbox Drive 2 Output Torque Limit
          Row[4]:
            Index = 3
            Value = 370.0
            Unit = Nm
            Description = Gearbox Drive 3 Output Torque Limit
          Row[5]:
            Index = 4
            Value = 17.0
            Unit = Nm
            Description = Gearbox Drive 4 Output Torque Limit
        CrossSectionLimits:
          Row[1]:
            Value = 4
            Unit = Variant
            Description = Type of dynamic model
          Row[2]:
            Index = 1
            Value = 10000.0
            Unit = N
            Description = 
          Row[3]:
            Index = 2
            Value = 10000.0
            Unit = N
            Description = 
          Row[4]:
            Index = 3
            Value = 10000.0
            Unit = N
            Description = 
          Row[5]:
            Index = 4
            Value = 141.0
            Unit = Nm
            Description = 
          Row[6]:
            Index = 5
            Value = 141.0
            Unit = Nm
            Description = 
          Row[7]:
            Index = 6
            Value = 10000.0
            Unit = Nm
            Description = 
          Row[8]:
            Index = 7
            Value = 750.0
            Unit = N
            Description = 
          Row[9]:
            Index = 8
            Value = 750.0
            Unit = N
            Description = 
          Row[10]:
            Index = 9
            Value = 750.0
            Unit = N
            Description = 
          Row[11]:
            Index = 10
            Value = 750.0
            Unit = N
            Description = 
          Row[12]:
            Index = 11
            Value = 750.0
            Unit = N
            Description = 
          Row[13]:
            Index = 12
            Value = 750.0
            Unit = N
            Description = 
      LoadDependentJerkLimitsIsReadOnly = 1
      LoadDependentJerkLimits = PayloadDependentJerkReduction
        JerkReduction[1]:
          PayloadInKgIsReadOnly = 1
          PayloadInKg = 0.0
          JerkReductionInPercentIsReadOnly = 1
          JerkReductionInPercent = 0.0
        JerkReduction[2]:
          PayloadInKgIsReadOnly = 1
          PayloadInKg = 7.0
          JerkReductionInPercentIsReadOnly = 1
          JerkReductionInPercent = 20.0
        JerkReduction[3]:
          PayloadInKgIsReadOnly = 1
          PayloadInKg = 13.0
          JerkReductionInPercentIsReadOnly = 1
          JerkReductionInPercent = 60.0
        JerkReduction[4]:
          PayloadInKgIsReadOnly = 1
          PayloadInKg = 19.0
          JerkReductionInPercentIsReadOnly = 1
          JerkReductionInPercent = 60.0
        JerkReduction[5]:
          PayloadInKgIsReadOnly = 1
          PayloadInKg = 23.0
          JerkReductionInPercentIsReadOnly = 1
          JerkReductionInPercent = 80.0
      JointAxesPositionLimits:
        JointAxisIsReadOnly = 1
        JointAxis[1]
        JointAxis[2]
        JointAxis[3]
        JointAxis[4]
      WorkingRangeIsReadOnly = 1
      WorkingRange = Extended
        MainCylinderDiameterIsReadOnly = 1
        MainCylinderDiameter = 1100.0
        BaseToTopConeIsReadOnly = 1
        BaseToTopCone = 735.0
        MainCylinderOffsetIsReadOnly = 1
        MainCylinderOffset = 270.0
        MainConeOffsetIsReadOnly = 1
        MainConeOffset = 350.0
        BottomConeOffsetIsReadOnly = 1
        BottomConeOffset = 420.0
        MainConeDiameterIsReadOnly = 1
        MainConeDiameter = 820.0
        BottomConeDiameterIsReadOnly = 1
        BottomConeDiameter = 340.0
        TopConeOffsetIsReadOnly = 1
        TopConeDiameterIsReadOnly = 1
        TopConeDiameter = 1100.0
```

### Config_8.axesgroupfeature - 5APC4100_TGL4_000/mappMotion/Robots/Codian_D4r1100R_2/Config_8.axesgroupfeature
```
Element Feature_TrkFrmSel_R2 (Type=axesgroupfeature)
  Type = TrackingFrameSelection
    Selectors:
      Selector[1]:
        Name = ProductSelector
        Strategy = MinimumDistanceToPoint
          Origin = MCS
            Translation:
              X = -300
              Z = 0
        Filters:
          Filter[1]:
            TrackingPathRef[1] = gTrkPath_Conveyor_1
          Filter[2] = SelectionArea
            Area[1] = Cylinder
              Origin = MCS
              Translation:
                X = -470
                Z = -100
              Dimensions:
                Radius = 475
                Height = 250
        LockingAfterSelection = AllSelectors
      Selector[2]:
        Name = PlacePositionSelector
        Strategy = MaximumXValueOnTrackingPath
        Filters:
          Filter[1]:
            TrackingPathRef[1] = gTrkPath_Conveyor_2
          Filter[2] = SelectionArea
            Area[1] = Cylinder
              Origin = MCS
              Translation:
                X = 250
                Z = -100
              Dimensions:
                Radius = 500
                Height = 250
          Filter[3] = SelectionArea
            Area[1] = Cylinder
              Origin = MCS
              Translation:
                Z = -100
              Dimensions:
                Radius = 450
                Height = 250
        LockingAfterSelection = AllSelectors
Element Feature_Programs_D4r1100R_2 (Type=axesgroupfeature)  // Codian D4-ST41-1100-R30 [RobotID="CodianD4ST41r1100R30" Version="6.4.1"]
  Type:
    InitialSettings:
      AccuracyHoldDelays = User defined
        UserAxesDelay = 0.06
    ProgramElements:
      PVs:
        PV[1]:
          PvName = ::MovePrg:GripperRobot2OpenClose
          Advanced:
            Alias = CloseGripper
            Synchronization = Path
Element Feature_Jogging_D4r1100R_2 (Type=axesgroupfeature)  // Codian D4-ST41-1100-R30 [RobotID="CodianD4ST41r1100R30" Version="6.4.1"]
  Type = Jogging
Element Feature_FeedForward_D4r1100R_2 (Type=axesgroupfeature)  // Codian D4-ST41-1100-R30 [RobotID="CodianD4ST41r1100R30" Version="6.4.1"]
  Type = FeedForward
    RiseTime = 0.25
    Filter = AxisJerkTime
```

### Config_10.axis - 5APC4100_TGL4_000/mappMotion/Robots/Codian_D4r1100R_3/Config_10.axis
```
Element gAxisQ1_D4r1100R_3 (Type=axis)  // Codian D4-ST41-1100-R30 [RobotID="CodianD4ST41r1100R30" Version="6.4.1"]
  BaseTypeIsReadOnly = 1
  BaseType = RotaryBounded
    MeasurementUnitIsReadOnly = 1
    MeasurementResolutionIsReadOnly = 1
    MeasurementResolution = 0.001
    CountDirectionIsReadOnly = 1
    CountDirection = Inverse
  MovementLimitsIsReadOnly = 1
  MovementLimits = InternalForPathControlledAxis
    Position:
      LowerLimitMin = -45.0
      UpperLimitMax = 103.0
      LowerLimit = -45.0
      UpperLimit = 103.0
    VelocityIsReadOnly = 1
    Velocity:
      VelocityMax = 410.0
      Velocity = 410.0
    AccelerationIsReadOnly = 1
    Acceleration:
      AccelerationMax = 25000.0
      Acceleration = 25000.0
    DecelerationIsReadOnly = 1
    Deceleration:
      DecelerationMax = 25000.0
      Deceleration = 25000.0
    JerkIsReadOnly = 1
    Jerk = Advanced
      JerkAccelerationPositiveMin = 0.0
      JerkAccelerationPositiveMax = 5000000.0
      JerkAccelerationPositive = 5000000.0
      JerkAccelerationNegativeMin = 0.0
      JerkAccelerationNegativeMax = 5000000.0
      JerkAccelerationNegative = 5000000.0
      JerkDecelerationPositiveMin = 0.0
      JerkDecelerationPositiveMax = 5000000.0
      JerkDecelerationPositive = 5000000.0
      JerkDecelerationNegativeMin = 0.0
      JerkDecelerationNegativeMax = 5000000.0
      JerkDecelerationNegative = 5000000.0
    TorqueIsReadOnly = 1
    Torque = Basic
      TorqueMax = 15.0
      Torque = 15.0
Element gAxisQ2_D4r1100R_3 (Type=axis)  // Codian D4-ST41-1100-R30 [RobotID="CodianD4ST41r1100R30" Version="6.4.1"]
  BaseTypeIsReadOnly = 1
  BaseType = RotaryBounded
    MeasurementUnitIsReadOnly = 1
    MeasurementResolutionIsReadOnly = 1
    MeasurementResolution = 0.001
    CountDirectionIsReadOnly = 1
    CountDirection = Inverse
  MovementLimitsIsReadOnly = 1
  MovementLimits = InternalForPathControlledAxis
    Position:
      LowerLimitMin = -45.0
      UpperLimitMax = 103.0
      LowerLimit = -45.0
      UpperLimit = 103.0
    VelocityIsReadOnly = 1
    Velocity:
      VelocityMax = 410.0
      Velocity = 410.0
    AccelerationIsReadOnly = 1
    Acceleration:
      AccelerationMax = 25000.0
      Acceleration = 25000.0
    DecelerationIsReadOnly = 1
    Deceleration:
      DecelerationMax = 25000.0
      Deceleration = 25000.0
    JerkIsReadOnly = 1
    Jerk = Advanced
      JerkAccelerationPositiveMin = 0.0
      JerkAccelerationPositiveMax = 5000000.0
      JerkAccelerationPositive = 5000000.0
      JerkAccelerationNegativeMin = 0.0
      JerkAccelerationNegativeMax = 5000000.0
      JerkAccelerationNegative = 5000000.0
      JerkDecelerationPositiveMin = 0.0
      JerkDecelerationPositiveMax = 5000000.0
      JerkDecelerationPositive = 5000000.0
      JerkDecelerationNegativeMin = 0.0
      JerkDecelerationNegativeMax = 5000000.0
      JerkDecelerationNegative = 5000000.0
    TorqueIsReadOnly = 1
    Torque = Basic
      TorqueMax = 15.0
      Torque = 15.0
Element gAxisQ3_D4r1100R_3 (Type=axis)  // Codian D4-ST41-1100-R30 [RobotID="CodianD4ST41r1100R30" Version="6.4.1"]
  BaseTypeIsReadOnly = 1
  BaseType = RotaryBounded
    MeasurementUnitIsReadOnly = 1
    MeasurementResolutionIsReadOnly = 1
    MeasurementResolution = 0.001
    CountDirectionIsReadOnly = 1
    CountDirection = Inverse
  MovementLimitsIsReadOnly = 1
  MovementLimits = InternalForPathControlledAxis
    Position:
      LowerLimitMin = -45.0
      UpperLimitMax = 103.0
      LowerLimit = -45.0
      UpperLimit = 103.0
    VelocityIsReadOnly = 1
    Velocity:
      VelocityMax = 410.0
      Velocity = 410.0
    AccelerationIsReadOnly = 1
    Acceleration:
      AccelerationMax = 25000.0
      Acceleration = 25000.0
    DecelerationIsReadOnly = 1
    Deceleration:
      DecelerationMax = 25000.0
      Deceleration = 25000.0
    JerkIsReadOnly = 1
    Jerk = Advanced
      JerkAccelerationPositiveMin = 0.0
      JerkAccelerationPositiveMax = 5000000.0
      JerkAccelerationPositive = 5000000.0
      JerkAccelerationNegativeMin = 0.0
      JerkAccelerationNegativeMax = 5000000.0
      JerkAccelerationNegative = 5000000.0
      JerkDecelerationPositiveMin = 0.0
      JerkDecelerationPositiveMax = 5000000.0
      JerkDecelerationPositive = 5000000.0
      JerkDecelerationNegativeMin = 0.0
      JerkDecelerationNegativeMax = 5000000.0
      JerkDecelerationNegative = 5000000.0
    TorqueIsReadOnly = 1
    Torque = Basic
      TorqueMax = 15.0
      Torque = 15.0
Element gAxisQC_D4r1100R_3 (Type=axis)  // Codian D4-ST41-1100-R30 [RobotID="CodianD4ST41r1100R30" Version="6.4.1"]
  BaseTypeIsReadOnly = 1
  BaseType = Rotary
    MeasurementUnitIsReadOnly = 1
    MeasurementResolutionIsReadOnly = 1
    MeasurementResolution = 0.001
    CountDirectionIsReadOnly = 1
  MovementLimitsIsReadOnly = 1
  MovementLimits = InternalForPathControlledAxis
    VelocityIsReadOnly = 1
    Velocity:
      VelocityMax = 1150.0
      Velocity = 1150.0
    AccelerationIsReadOnly = 1
    Acceleration:
      AccelerationMax = 28000.0
      Acceleration = 28000.0
    DecelerationIsReadOnly = 1
    Deceleration:
      DecelerationMax = 28000.0
      Deceleration = 28000.0
    JerkIsReadOnly = 1
    Jerk = Advanced
      JerkAccelerationPositiveMin = 0.0
      JerkAccelerationPositiveMax = 4000000.0
      JerkAccelerationPositive = 4000000.0
      JerkAccelerationNegativeMin = 0.0
      JerkAccelerationNegativeMax = 4000000.0
      JerkAccelerationNegative = 4000000.0
      JerkDecelerationPositiveMin = 0.0
      JerkDecelerationPositiveMax = 4000000.0
      JerkDecelerationPositive = 4000000.0
      JerkDecelerationNegativeMin = 0.0
      JerkDecelerationNegativeMax = 4000000.0
      JerkDecelerationNegative = 4000000.0
    TorqueIsReadOnly = 1
    Torque = Basic
      TorqueMax = 9.0
      Torque = 9.0
```

### Config_11.mechanicalsystem - 5APC4100_TGL4_000/mappMotion/Robots/Codian_D4r1100R_3/Config_11.mechanicalsystem
```
Element MechSys_D4r1100R_3 (Type=mechanicalsystem)  // Codian D4-ST41-1100-R30 [RobotID="CodianD4ST41r1100R30" Version="6.4.1"]
  TypeIsReadOnly = 1
  Type = Delta
    SubtypeIsReadOnly = 1
    Subtype = 4AxesDeltaA
      SceneViewerObject = ObjectID
        ID = 2540
      DescriptionIsReadOnly = 1
      Description:
        Dimensions:
          BasePlatform:
            ArmLinkPointIsReadOnly = 1
            Arm1LinkPoint:
              Radius = 207.5
              Z = -110.0
            Arm2LinkPoint:
              Angle = -120.0
              Radius = 207.5
              Z = -110.0
            Arm3LinkPoint:
              Angle = -240.0
              Radius = 207.5
              Z = -110.0
          Arms:
            ArmIsReadOnly = 1
            Arm1:
              UpperArmLength = 320.0
              LowerArmLength = 850.0
            Arm2:
              UpperArmLength = 320.0
              LowerArmLength = 850.0
            Arm3:
              UpperArmLength = 320.0
              LowerArmLength = 850.0
            LowerArmPairDistance = 154.0
          EndEffectorPlatform:
            ArmLinkPointIsReadOnly = 1
            Arm1LinkPoint:
              Radius = 70.0
            Arm2LinkPoint:
              Radius = 70.0
            Arm3LinkPoint:
              Radius = 70.0
            TranslationToFlange:
              Z = -59.0
        Offsets:
          JointAxisIsReadOnly = 1
          JointAxis[1]
          JointAxis[2]
          JointAxis[3]
          JointAxis[4]
        CountDirections:
          JointAxisIsReadOnly = 1
          JointAxis[1]
          JointAxis[2]
          JointAxis[3]
          JointAxis[4]
      TcpOrientation:
        Frames = Used
      WireFrameModel:
        UpperArm1:
          Distance = 5
        LowerArm1:
          Distance = 5
        UpperArm2:
          Distance = 5
        LowerArm2:
          Distance = 5
        UpperArm3:
          Distance = 5
        LowerArm3:
          Distance = 5
        EndEffectorPlatformToFlange:
          Distance = 5
        FlangeToTcp = NotUsed
      DynamicModelIsReadOnly = 1
      InternalDynamicModelIsReadOnly = 1
      InternalDynamicModel = Used
        TypeIsReadOnly = 1
        Type = Codian D4-ST41-1100-R30
        Row[1]:
          Value = 4
          Unit = Variant
          Description = Type of dynamic model
        Row[2]:
          Index = 1
          Value = 2.739
          Unit = 
          Description = m1
        Row[3]:
          Index = 2
          Value = 0.2990988
          Unit = 
          Description = m1*rc1x
        Row[4]:
          Index = 3
          Unit = 
          Description = m1*rc1y
        Row[5]:
          Index = 4
          Value = 0.0257466
          Unit = 
          Description = m1*rc1z
        Row[6]:
          Index = 5
          Unit = 
          Description = m1*rc1x*rc1y
        Row[7]:
          Index = 6
          Unit = 
          Description = m1*rc1y*rc1z
        Row[8]:
          Index = 7
          Value = 0.00281152872
          Unit = 
          Description = m1*rc1x*rc1z
        Row[9]:
          Index = 8
          Value = 0.03266158896
          Unit = 
          Description = m1*rc1x^2
        Row[10]:
          Index = 9
          Unit = 
          Description = m1*rc1y^2
        Row[11]:
          Index = 10
          Value = 0.00024201804
          Unit = 
          Description = m1*rc1z^2
        Row[12]:
          Index = 11
          Unit = 
          Description = Jxx1
        Row[13]:
          Index = 12
          Value = 0.0423
          Unit = 
          Description = Jyy1
        Row[14]:
          Index = 13
          Unit = 
          Description = Jzz1
        Row[15]:
          Index = 14
          Value = 2.739
          Unit = 
          Description = m2
        Row[16]:
          Index = 15
          Value = 0.2990988
          Unit = 
          Description = m2*rc2x
        Row[17]:
          Index = 16
          Unit = 
          Description = m2*rc2y
        Row[18]:
          Index = 17
          Value = 0.0257466
          Unit = 
          Description = m2*rc2z
        Row[19]:
          Index = 18
          Unit = 
          Description = m2*rc2x*rc2y
        Row[20]:
          Index = 19
          Unit = 
          Description = m2*rc2y*rc2z
        Row[21]:
          Index = 20
          Value = 0.00281152872
          Unit = 
          Description = m2*rc2x*rc2z
        Row[22]:
          Index = 21
          Value = 0.03266158896
          Unit = 
          Description = m2*rc2x^2
        Row[23]:
          Index = 22
          Unit = 
          Description = m2*rc2y^2
        Row[24]:
          Index = 23
          Value = 0.00024201804
          Unit = 
          Description = m2*rc2z^2
        Row[25]:
          Index = 24
          Unit = 
          Description = Jxx2
        Row[26]:
          Index = 25
          Value = 0.0423
          Unit = 
          Description = Jyy2
        Row[27]:
          Index = 26
          Unit = 
          Description = Jzz2
        Row[28]:
          Index = 27
          Value = 2.739
          Unit = 
          Description = m3
        Row[29]:
          Index = 28
          Value = 0.2990988
          Unit = 
          Description = m3*rc3x
        Row[30]:
          Index = 29
          Unit = 
          Description = m3*rc3y
        Row[31]:
          Index = 30
          Value = 0.0257466
          Unit = 
          Description = m3*rc3z
        Row[32]:
          Index = 31
          Unit = 
          Description = m3*rc3x*rc3y
        Row[33]:
          Index = 32
          Unit = 
          Description = m3*rc3y*rc3z
        Row[34]:
          Index = 33
          Value = 0.00281152872
          Unit = 
          Description = m3*rc3x*rc3z
        Row[35]:
          Index = 34
          Value = 0.03266158896
          Unit = 
          Description = m3*rc3x^2
        Row[36]:
          Index = 35
          Unit = 
          Description = m3*rc3y^2
        Row[37]:
          Index = 36
          Value = 0.00024201804
          Unit = 
          Description = m3*rc3z^2
        Row[38]:
          Index = 37
          Unit = 
          Description = Jxx3
        Row[39]:
          Index = 38
          Value = 0.0423
          Unit = 
          Description = Jyy3
        Row[40]:
          Index = 39
          Unit = 
          Description = Jzz3
        Row[41]:
          Index = 40
          Value = 0.808
          Unit = 
          Description = m4
        Row[42]:
          Index = 41
          Unit = 
          Description = m4*rc4x
        Row[43]:
          Index = 42
          Unit = 
          Description = m4*rc4y
        Row[44]:
          Index = 43
          Unit = 
          Description = m4*rc4z
        Row[45]:
          Index = 44
          Unit = 
          Description = m4*rc4x*rc4y
        Row[46]:
          Index = 45
          Unit = 
          Description = m4*rc4y*rc4z
        Row[47]:
          Index = 46
          Unit = 
          Description = m4*rc4x*rc4z
        Row[48]:
          Index = 47
          Unit = 
          Description = m4*rc4x^2
        Row[49]:
          Index = 48
          Unit = 
          Description = m4*rc4y^2
        Row[50]:
          Index = 49
          Unit = 
          Description = m4*rc4z^2
        Row[51]:
          Index = 50
          Value = 0.0901
          Unit = 
          Description = Jxx4
        Row[52]:
          Index = 51
          Value = 0.0901
          Unit = 
          Description = Jyy4
        Row[53]:
          Index = 52
          Unit = 
          Description = Jzz4
        Row[54]:
          Index = 53
          Value = 0.808
          Unit = 
          Description = m5
        Row[55]:
          Index = 54
          Unit = 
          Description = m5*rc5x
        Row[56]:
          Index = 55
          Unit = 
          Description = m5*rc5y
        Row[57]:
          Index = 56
          Unit = 
          Description = m5*rc5z
        Row[58]:
          Index = 57
          Unit = 
          Description = m5*rc5x*rc5y
        Row[59]:
          Index = 58
          Unit = 
          Description = m5*rc5y*rc5z
        Row[60]:
          Index = 59
          Unit = 
          Description = m5*rc5x*rc5z
        Row[61]:
          Index = 60
          Unit = 
          Description = m5*rc5x^2
        Row[62]:
          Index = 61
          Unit = 
          Description = m5*rc5y^2
        Row[63]:
          Index = 62
          Unit = 
          Description = m5*rc5z^2
        Row[64]:
          Index = 63
          Value = 0.0901
          Unit = 
          Description = Jxx5
        Row[65]:
          Index = 64
          Value = 0.0901
          Unit = 
          Description = Jyy5
        Row[66]:
          Index = 65
          Unit = 
          Description = Jzz5
        Row[67]:
          Index = 66
          Value = 0.808
          Unit = 
          Description = m6
        Row[68]:
          Index = 67
          Unit = 
          Description = m6*rc6x
        Row[69]:
          Index = 68
          Unit = 
          Description = m6*rc6y
        Row[70]:
          Index = 69
          Unit = 
          Description = m6*rc6z
        Row[71]:
          Index = 70
          Unit = 
          Description = m6*rc6x*rc6y
        Row[72]:
          Index = 71
          Unit = 
          Description = m6*rc6y*rc6z
        Row[73]:
          Index = 72
          Unit = 
          Description = m6*rc6x*rc6z
        Row[74]:
          Index = 73
          Unit = 
          Description = m6*rc6x^2
        Row[75]:
          Index = 74
          Unit = 
          Description = m6*rc6y^2
        Row[76]:
          Index = 75
          Unit = 
          Description = m6*rc6z^2
        Row[77]:
          Index = 76
          Value = 0.0901
          Unit = 
          Description = Jxx6
        Row[78]:
          Index = 77
          Value = 0.0901
          Unit = 
          Description = Jyy6
        Row[79]:
          Index = 78
          Unit = 
          Description = Jzz6
        Row[80]:
          Index = 79
          Value = 2.005
          Unit = 
          Description = m7
        Row[81]:
          Index = 80
          Unit = 
          Description = m7*rc7x
        Row[82]:
          Index = 81
          Unit = 
          Description = m7*rc7y
        Row[83]:
          Index = 82
          Value = 0.47159605
          Unit = 
          Description = m7*rc7z
        Row[84]:
          Index = 83
          Unit = 
          Description = m7*rc7x*rc7y
        Row[85]:
          Index = 84
          Unit = 
          Description = m7*rc7y*rc7z
        Row[86]:
          Index = 85
          Unit = 
          Description = m7*rc7x*rc7z
        Row[87]:
          Index = 86
          Unit = 
          Description = m7*rc7x^2
        Row[88]:
          Index = 87
          Unit = 
          Description = m7*rc7y^2
        Row[89]:
          Index = 88
          Value = 0.110924106921
          Unit = 
          Description = m7*rc7z^2
        Row[90]:
          Index = 89
          Value = 0.071421443
          Unit = 
          Description = Jxx7
        Row[91]:
          Index = 90
          Value = 0.071421443
          Unit = 
          Description = Jyy7
        Row[92]:
          Index = 91
          Value = 0.0003844
          Unit = 
          Description = Jzz7
        Row[93]:
          Index = 92
          Value = 1.8
          Unit = 
          Description = m8
        Row[94]:
          Index = 93
          Unit = 
          Description = m8*rc8x
        Row[95]:
          Index = 94
          Unit = 
          Description = m8*rc8y
        Row[96]:
          Index = 95
          Value = 0.520488
          Unit = 
          Description = m8*rc8z
        Row[97]:
          Index = 96
          Unit = 
          Description = m8*rc8x*rc8y
        Row[98]:
          Index = 97
          Unit = 
          Description = m8*rc8y*rc8z
        Row[99]:
          Index = 98
          Unit = 
          Description = m8*rc8x*rc8z
        Row[100]:
          Index = 99
          Unit = 
          Description = m8*rc8x^2
        Row[101]:
          Index = 100
          Unit = 
          Description = m8*rc8y^2
        Row[102]:
          Index = 101
          Value = 0.15050431008
          Unit = 
          Description = m8*rc8z^2
        Row[103]:
          Index = 102
          Value = 0.093006951
          Unit = 
          Description = Jxx8
        Row[104]:
          Index = 103
          Value = 0.093006951
          Unit = 
          Description = Jyy8
        Row[105]:
          Index = 104
          Value = 0.00097
          Unit = 
          Description = Jzz8
        Row[106]:
          Index = 105
          Value = 2.094
          Unit = 
          Description = m9
        Row[107]:
          Index = 106
          Unit = 
          Description = m9*rc9x
        Row[108]:
          Index = 107
          Unit = 
          Description = m9*rc9y
        Row[109]:
          Index = 108
          Unit = 
          Description = m9*rc9z
        Row[110]:
          Index = 109
          Unit = 
          Description = m9*rc9x*rc9y
        Row[111]:
          Index = 110
          Unit = 
          Description = m9*rc9y*rc9z
        Row[112]:
          Index = 111
          Unit = 
          Description = m9*rc9x*rc9z
        Row[113]:
          Index = 112
          Unit = 
          Description = m9*rc9x^2
        Row[114]:
          Index = 113
          Unit = 
          Description = m9*rc9y^2
        Row[115]:
          Index = 114
          Unit = 
          Description = m9*rc9z^2
        Row[116]:
          Index = 115
          Unit = 
          Description = Jxx9
        Row[117]:
          Index = 116
          Unit = 
          Description = Jyy9
        Row[118]:
          Index = 117
          Unit = 
          Description = Jzz9
        Row[119]:
          Index = 118
          Unit = 
          Description = m10
        Row[120]:
          Index = 119
          Unit = 
          Description = m10*rc10x
        Row[121]:
          Index = 120
          Unit = 
          Description = m10*rc10y
        Row[122]:
          Index = 121
          Unit = 
          Description = m10*rc10z
        Row[123]:
          Index = 122
          Unit = 
          Description = m10*rc10x*rc10y
        Row[124]:
          Index = 123
          Unit = 
          Description = m10*rc10y*rc10z
        Row[125]:
          Index = 124
          Unit = 
          Description = m10*rc10x*rc10z
        Row[126]:
          Index = 125
          Unit = 
          Description = m10*rc10x^2
        Row[127]:
          Index = 126
          Unit = 
          Description = m10*rc10y^2
        Row[128]:
          Index = 127
          Unit = 
          Description = m10*rc10z^2
        Row[129]:
          Index = 128
          Unit = 
          Description = Jxx10
        Row[130]:
          Index = 129
          Unit = 
          Description = Jyy10
        Row[131]:
          Index = 130
          Value = 0.0001507
          Unit = 
          Description = Jzz10
        Row[132]:
          Index = 144
          Value = 0.0005703
          Unit = 
          Description = JDrive1
        Row[133]:
          Index = 145
          Value = 0.0005703
          Unit = 
          Description = JDrive2
        Row[134]:
          Index = 146
          Value = 0.0005703
          Unit = 
          Description = JDrive3
        Row[135]:
          Index = 147
          Value = 0.0001462
          Unit = 
          Description = JDrive4
        Row[136]:
          Index = 148
          Value = 2.35907414398
          Unit = 
          Description = dV1
        Row[137]:
          Index = 149
          Value = 2.35907414398
          Unit = 
          Description = dV2
        Row[138]:
          Index = 150
          Value = 2.35907414398
          Unit = 
          Description = dV3
        Row[139]:
          Index = 151
          Value = 0.0159154943092
          Unit = 
          Description = dV4
        Row[140]:
          Index = 152
          Value = 4.235
          Unit = 
          Description = dC1
        Row[141]:
          Index = 153
          Value = 4.235
          Unit = 
          Description = dC2
        Row[142]:
          Index = 154
          Value = 4.235
          Unit = 
          Description = dC3
        Row[143]:
          Index = 155
          Value = 1.0
          Unit = 
          Description = dC4
      InternalDynamicLimits = Used
        TypeIsReadOnly = 1
        Type = Codian D4-ST41-1100-R30
        GearboxLimits:
          Row[1]:
            Value = 4
            Unit = Variant
            Description = Type of dynamic model
          Row[2]:
            Index = 1
            Value = 370.0
            Unit = Nm
            Description = Gearbox Drive 1 Output Torque Limit
          Row[3]:
            Index = 2
            Value = 370.0
            Unit = Nm
            Description = Gearbox Drive 2 Output Torque Limit
          Row[4]:
            Index = 3
            Value = 370.0
            Unit = Nm
            Description = Gearbox Drive 3 Output Torque Limit
          Row[5]:
            Index = 4
            Value = 17.0
            Unit = Nm
            Description = Gearbox Drive 4 Output Torque Limit
        CrossSectionLimits:
          Row[1]:
            Value = 4
            Unit = Variant
            Description = Type of dynamic model
          Row[2]:
            Index = 1
            Value = 10000.0
            Unit = N
            Description = 
          Row[3]:
            Index = 2
            Value = 10000.0
            Unit = N
            Description = 
          Row[4]:
            Index = 3
            Value = 10000.0
            Unit = N
            Description = 
          Row[5]:
            Index = 4
            Value = 141.0
            Unit = Nm
            Description = 
          Row[6]:
            Index = 5
            Value = 141.0
            Unit = Nm
            Description = 
          Row[7]:
            Index = 6
            Value = 10000.0
            Unit = Nm
            Description = 
          Row[8]:
            Index = 7
            Value = 750.0
            Unit = N
            Description = 
          Row[9]:
            Index = 8
            Value = 750.0
            Unit = N
            Description = 
          Row[10]:
            Index = 9
            Value = 750.0
            Unit = N
            Description = 
          Row[11]:
            Index = 10
            Value = 750.0
            Unit = N
            Description = 
          Row[12]:
            Index = 11
            Value = 750.0
            Unit = N
            Description = 
          Row[13]:
            Index = 12
            Value = 750.0
            Unit = N
            Description = 
      LoadDependentJerkLimitsIsReadOnly = 1
      LoadDependentJerkLimits = PayloadDependentJerkReduction
        JerkReduction[1]:
          PayloadInKgIsReadOnly = 1
          PayloadInKg = 0.0
          JerkReductionInPercentIsReadOnly = 1
          JerkReductionInPercent = 0.0
        JerkReduction[2]:
          PayloadInKgIsReadOnly = 1
          PayloadInKg = 7.0
          JerkReductionInPercentIsReadOnly = 1
          JerkReductionInPercent = 20.0
        JerkReduction[3]:
          PayloadInKgIsReadOnly = 1
          PayloadInKg = 13.0
          JerkReductionInPercentIsReadOnly = 1
          JerkReductionInPercent = 60.0
        JerkReduction[4]:
          PayloadInKgIsReadOnly = 1
          PayloadInKg = 19.0
          JerkReductionInPercentIsReadOnly = 1
          JerkReductionInPercent = 60.0
        JerkReduction[5]:
          PayloadInKgIsReadOnly = 1
          PayloadInKg = 23.0
          JerkReductionInPercentIsReadOnly = 1
          JerkReductionInPercent = 80.0
      JointAxesPositionLimits:
        JointAxisIsReadOnly = 1
        JointAxis[1]
        JointAxis[2]
        JointAxis[3]
        JointAxis[4]
      WorkingRangeIsReadOnly = 1
      WorkingRange = Extended
        MainCylinderDiameterIsReadOnly = 1
        MainCylinderDiameter = 1100.0
        BaseToTopConeIsReadOnly = 1
        BaseToTopCone = 735.0
        MainCylinderOffsetIsReadOnly = 1
        MainCylinderOffset = 270.0
        MainConeOffsetIsReadOnly = 1
        MainConeOffset = 350.0
        BottomConeOffsetIsReadOnly = 1
        BottomConeOffset = 420.0
        MainConeDiameterIsReadOnly = 1
        MainConeDiameter = 820.0
        BottomConeDiameterIsReadOnly = 1
        BottomConeDiameter = 340.0
        TopConeOffsetIsReadOnly = 1
        TopConeDiameterIsReadOnly = 1
        TopConeDiameter = 1100.0
```

### Config_12.axesgroupfeature - 5APC4100_TGL4_000/mappMotion/Robots/Codian_D4r1100R_3/Config_12.axesgroupfeature
```
Element Feature_Programs_D4r1100R_3 (Type=axesgroupfeature)  // Codian D4-ST41-1100-R30 [RobotID="CodianD4ST41r1100R30" Version="6.4.1"]
  Type:
    InitialSettings:
      AccuracyHoldDelays = User defined
        UserAxesDelay = 0.06
    ProgramElements:
      PVs:
        PV[1]:
          PvName = ::MovePrg:GripperRobot3OpenClose
          Advanced:
            Alias = CloseGripper
            Synchronization = Path
Element Feature_Jogging_D4r1100R_3 (Type=axesgroupfeature)  // Codian D4-ST41-1100-R30 [RobotID="CodianD4ST41r1100R30" Version="6.4.1"]
  Type = Jogging
Element Feature_FeedForward_D4r1100R_3 (Type=axesgroupfeature)  // Codian D4-ST41-1100-R30 [RobotID="CodianD4ST41r1100R30" Version="6.4.1"]
  Type = FeedForward
    RiseTime = 0.25
    Filter = AxisJerkTime
```
